FUNCTION_BLOCK ABSTRACT OpcUaRequestItem EXTENDS TC.ToolkitObject
VAR
	_ConnectionHandle : DWORD;
END_VAR

METHOD ABSTRACT GetHandle : OPC_UA_ACTION_EXECUTION_STATE
VAR_INPUT
	connectionHandle : DWORD;
END_VAR
VAR_OUTPUT
	exception : Exception;
END_VAR
END_METHOD

METHOD ABSTRACT PerformAction : OPC_UA_ACTION_EXECUTION_STATE
VAR_OUTPUT
	exception : Exception;
END_VAR
END_METHOD

METHOD ABSTRACT ReleaseHandle : OPC_UA_ACTION_EXECUTION_STATE
VAR_OUTPUT
	exception : Exception;
END_VAR
END_METHOD

METHOD ABSTRACT Reset
END_METHOD

METHOD ABSTRACT ResetAction
END_METHOD

METHOD ABSTRACT SetNamespaceIndexForNamespaceUri
VAR_INPUT
	namespaceUri : STRING(Tc2_System.MAX_STRING_LENGTH);
	namespaceIndex : UINT;
END_VAR
END_METHOD

END_FUNCTION_BLOCK

(* stored: Version 1.1.0.1
   POU OpcUaRequestItem: Id {200666ba-908b-472f-8c22-3b6d239e05af}, SpecialFunc None
   Method GetHandle: Id {805f5ab9-be9e-4e41-b4ea-701990c1f4fa}
   Method PerformAction: Id {a12b7ee3-b79d-445f-9ad0-7179931cf62e}
   Method ReleaseHandle: Id {3ff0446a-2f58-4162-96ed-d000835983a0}
   Method Reset: Id {c5f8ea59-0268-4c4a-a1c2-551dd982ac25}
   Method ResetAction: Id {5fd04d9a-1dea-46bb-9f6e-0666366f1d1d}
   Method SetNamespaceIndexForNamespaceUri: Id {c5a5d65d-1db4-4820-ba1f-dfb2ee3f577a} *)
